{attribute 'pack_mode' := '1'}
TYPE ST_ShutterStatus EXTENDS ST_PLCMsg:
STRUCT
    nMotionProfile: DINT; (* Motion profile index. *)
    bIsCalibrated: BOOL;
    nSmState: DINT;
    stAxis: ARRAY [0..1] OF ST_AxisStatus;
END_STRUCT
END_TYPE

(* stored: Version 1.1.0.1, ProductVersion 3.1.4022.18
   DUT ST_ShutterStatus: Id {92b4458d-b7e8-4988-b98b-43af5ff05814} *)
